FUNCTION F_ValidateRequester : E_RpcMethodResponse
VAR_INPUT
    eRequester        : E_Requester;
    bSourceLocked     : BOOL;
    bFaulted          : BOOL;
    bAllowWhenFaulted : BOOL;
    bSkipSourceCheck  : BOOL;
END_VAR

IF NOT bSkipSourceCheck AND bSourceLocked AND eRequester = E_Requester.OPERATOR THEN
    F_ValidateRequester := E_RpcMethodResponse.REJECTED_SOURCE_NOT_ALLOWED;
ELSIF bFaulted AND NOT bAllowWhenFaulted THEN
    F_ValidateRequester := E_RpcMethodResponse.REJECTED_FAULTED;
ELSE
    F_ValidateRequester := E_RpcMethodResponse.ACCEPTED;
END_IF;

END_FUNCTION

(* stored: Version 1.1.0.1, ProductVersion 3.1.4026.12
   POU F_ValidateRequester: Id {b1234567-1234-1234-1234-12345678C001}, SpecialFunc None *)
